// TIA Portal V17 export
// export: Created 2023-02-13T11:16:21.0492472Z, ExportSetting WithDefaults, DisplayName Totally Integrated Automation Portal, DisplayVersion V17, DisplayName TIA Portal Openness, DisplayVersion V17, DisplayName TIA Portal Teamcenter Gateway, DisplayVersion V17, DisplayName TIA Portal Version Control Interface, DisplayVersion V17, DisplayName SINAMICS Startdrive Advanced, DisplayVersion V17, DisplayName SINAMICS Startdrive G130, G150, S120, S150, SINAMICS MV, S210, DisplayVersion V17, DisplayName SINAMICS Startdrive G110M, G120, G120C, G120D, G120P, G115D, DisplayVersion V17, DisplayName STEP 7 Professional, DisplayVersion V17, DisplayName STEP 7 Safety, DisplayVersion V17, DisplayName WinCC Professional, DisplayVersion V17
DATA_BLOCK "IO_Valve_Blending_DB"   // DB8
VERSION : 0.1
// stored: AutoNumber true, DBAccessibleFromOPCUA true, DBAccessibleFromWebserver true, InstanceOfName IO_Valve_Blending, InstanceOfType FB
"IO_Valve_Blending"
   // VAR_INPUT
   //    lock : Bool;
   //    Init : Bool;
   //    Reset : Bool;
   // END_VAR
   // VAR
   //    "AV-20.01" { S7_SetPoint := 'True'} : "Valve";
   //    "AV-20.02" { S7_SetPoint := 'True'} : "Valve";
   //    "AV-20.03" { S7_SetPoint := 'True'} : "Valve";
   //    "AV-20.04" { S7_SetPoint := 'True'} : "Valve";
   //    "AV-20.05" { S7_SetPoint := 'True'} : "Valve";
   //    "AV-20.06" { S7_SetPoint := 'True'} : "Valve";
   //    "AV-20.07" { S7_SetPoint := 'True'} : "Valve";
   //    "AV-20.08" { S7_SetPoint := 'True'} : "Valve";
   //    "AV-20.09" { S7_SetPoint := 'True'} : "Valve";
   //    "AV-20.10" { S7_SetPoint := 'True'} : "Valve";
   //    "AV-20.11" { S7_SetPoint := 'True'} : "Valve";
   //    "AV-20.12" { S7_SetPoint := 'True'} : "Valve";
   //    "AV-20.13" { S7_SetPoint := 'True'} : "Valve";
   //    "AV-20.14" { S7_SetPoint := 'True'} : "Valve";
   //    "AV-20.15" { S7_SetPoint := 'True'} : "Valve";
   //    "AV-20.16" { S7_SetPoint := 'True'} : "Valve";
   //    "AV-20.17" { S7_SetPoint := 'True'} : "Valve";
   //    "AV-20.31" { S7_SetPoint := 'True'} : "Valve";
   //    "AV-20.32" { S7_SetPoint := 'True'} : "Valve";
   //    "AV-20.33" { S7_SetPoint := 'True'} : "Valve";
   //    "AV-20.34" { S7_SetPoint := 'True'} : "Valve";
   //    "AV-20.35" { S7_SetPoint := 'True'} : "Valve";
   //    "AV-20.36" { S7_SetPoint := 'True'} : "Valve";
   //    "AV-20.37" { S7_SetPoint := 'True'} : "Valve";
   //    "AV-20.38" { S7_SetPoint := 'True'} : "Valve";
   //    "AV-20.39" { S7_SetPoint := 'True'} : "Valve";
   //    "AV-20.40" { S7_SetPoint := 'True'} : "Valve";
   //    "AV-20.41" { S7_SetPoint := 'True'} : "Valve";
   //    "AV-21.01" { S7_SetPoint := 'True'} : "Valve";
   //    "AV-21.02" { S7_SetPoint := 'True'} : "Valve";
   //    "AV-21.03" { S7_SetPoint := 'True'} : "Valve";
   //    "AV-21.04" { S7_SetPoint := 'True'} : "Valve";
   //    "AV-21.05" { S7_SetPoint := 'True'} : "Valve";
   //    "AV-21.06" { S7_SetPoint := 'True'} : "Valve";
   //    "AV-21.07" { S7_SetPoint := 'True'} : "Valve";
   //    "AV-21.08" { S7_SetPoint := 'True'} : "Valve";
   //    "AV-21.09" { S7_SetPoint := 'True'} : "Valve";
   //    "AV-21.10" { S7_SetPoint := 'True'} : "Valve";
   //    "AV-21.11" { S7_SetPoint := 'True'} : "Valve";
   //    "AV-21.12" { S7_SetPoint := 'True'} : "Valve";
   //    "AV-21.13" { S7_SetPoint := 'True'} : "Valve";
   //    "AV-21.14" { S7_SetPoint := 'True'} : "Valve";
   //    "AV-21.15" { S7_SetPoint := 'True'} : "Valve";
   //    "AV-21.16" { S7_SetPoint := 'True'} : "Valve";
   //    "AV-21.17" { S7_SetPoint := 'True'} : "Valve";
   //    "AV-21.18" { S7_SetPoint := 'True'} : "Valve";
   //    "AV-21.31" { S7_SetPoint := 'True'} : "Valve";
   //    "AV-21.32" { S7_SetPoint := 'True'} : "Valve";
   //    "AV-21.33" { S7_SetPoint := 'True'} : "Valve";
   //    "AV-21.34" { S7_SetPoint := 'True'} : "Valve";
   //    "AV-21.35" { S7_SetPoint := 'True'} : "Valve";
   //    "AV-21.36" { S7_SetPoint := 'True'} : "Valve";
   //    "AV-21.37" { S7_SetPoint := 'True'} : "Valve";
   //    "AV-21.38" { S7_SetPoint := 'True'} : "Valve";
   //    "AV-21.39" { S7_SetPoint := 'True'} : "Valve";
   //    "AV-21.40" { S7_SetPoint := 'True'} : "Valve";
   //    "AV-21.41" { S7_SetPoint := 'True'} : "Valve";
   //    "AV-22.01" { S7_SetPoint := 'True'} : "Valve";
   //    "AV-22.02" { S7_SetPoint := 'True'} : "Valve";
   //    "AV-22.03" { S7_SetPoint := 'True'} : "Valve";
   //    "AV-22.06" { S7_SetPoint := 'True'} : "Valve";
   //    "AV-22.11" { S7_SetPoint := 'True'} : "Valve";
   //    "AV-22.21" { S7_SetPoint := 'True'} : "Valve";
   //    "AV-22.22" { S7_SetPoint := 'True'} : "Valve";
   //    "AV-30.01" { S7_SetPoint := 'True'} : "Valve";
   //    "AV-30.02" { S7_SetPoint := 'True'} : "Valve";
   //    "AV-30.03" { S7_SetPoint := 'True'} : "Valve";
   //    "AV-30.04" { S7_SetPoint := 'True'} : "Valve";
   //    "AV-30.05" { S7_SetPoint := 'True'} : "Valve";
   //    "AV-30.06" { S7_SetPoint := 'True'} : "Valve";
   //    "AV-30.07" { S7_SetPoint := 'True'} : "Valve";
   //    "AV-30.08" { S7_SetPoint := 'True'} : "Valve";
   //    "AV-30.09" { S7_SetPoint := 'True'} : "Valve";
   //    "AV-30.10" { S7_SetPoint := 'True'} : "Valve";
   //    "AV-30.11" { S7_SetPoint := 'True'} : "Valve";
   //    "AV-30.12" { S7_SetPoint := 'True'} : "Valve";
   //    "AV-30.13" { S7_SetPoint := 'True'} : "Valve";
   //    "AV-30.14" { S7_SetPoint := 'True'} : "Valve";
   //    "AV-30.15" { S7_SetPoint := 'True'} : "Valve";
   //    "AV-30.16" { S7_SetPoint := 'True'} : "Valve";
   //    "AV-30.17" { S7_SetPoint := 'True'} : "Valve";
   //    "AV-30.31" { S7_SetPoint := 'True'} : "Valve";
   //    "AV-30.32" { S7_SetPoint := 'True'} : "Valve";
   //    "AV-30.33" { S7_SetPoint := 'True'} : "Valve";
   //    "AV-30.34" { S7_SetPoint := 'True'} : "Valve";
   //    "AV-30.35" { S7_SetPoint := 'True'} : "Valve";
   //    "AV-30.36" { S7_SetPoint := 'True'} : "Valve";
   //    "AV-30.37" { S7_SetPoint := 'True'} : "Valve";
   //    "AV-30.38" { S7_SetPoint := 'True'} : "Valve";
   //    "AV-30.39" { S7_SetPoint := 'True'} : "Valve";
   //    "AV-30.40" { S7_SetPoint := 'True'} : "Valve";
   //    "AV-30.41" { S7_SetPoint := 'True'} : "Valve";
   //    "AV-31.01" { S7_SetPoint := 'True'} : "Valve";
   //    "AV-31.02" { S7_SetPoint := 'True'} : "Valve";
   //    "AV-31.03" { S7_SetPoint := 'True'} : "Valve";
   //    "AV-31.04" { S7_SetPoint := 'True'} : "Valve";
   //    "AV-31.05" { S7_SetPoint := 'True'} : "Valve";
   //    "AV-31.06" { S7_SetPoint := 'True'} : "Valve";
   //    "AV-31.07" { S7_SetPoint := 'True'} : "Valve";
   //    "AV-31.08" { S7_SetPoint := 'True'} : "Valve";
   //    "AV-31.09" { S7_SetPoint := 'True'} : "Valve";
   //    "AV-31.10" { S7_SetPoint := 'True'} : "Valve";
   //    "AV-31.11" { S7_SetPoint := 'True'} : "Valve";
   //    "AV-31.12" { S7_SetPoint := 'True'} : "Valve";
   //    "AV-31.13" { S7_SetPoint := 'True'} : "Valve";
   //    "AV-31.14" { S7_SetPoint := 'True'} : "Valve";
   //    "AV-31.15" { S7_SetPoint := 'True'} : "Valve";
   //    "AV-31.16" { S7_SetPoint := 'True'} : "Valve";
   //    "AV-31.17" { S7_SetPoint := 'True'} : "Valve";
   //    "AV-31.18" { S7_SetPoint := 'True'} : "Valve";
   //    "AV-31.31" { S7_SetPoint := 'True'} : "Valve";
   //    "AV-31.32" { S7_SetPoint := 'True'} : "Valve";
   //    "AV-31.33" { S7_SetPoint := 'True'} : "Valve";
   //    "AV-31.34" { S7_SetPoint := 'True'} : "Valve";
   //    "AV-31.35" { S7_SetPoint := 'True'} : "Valve";
   //    "AV-31.36" { S7_SetPoint := 'True'} : "Valve";
   //    "AV-31.37" { S7_SetPoint := 'True'} : "Valve";
   //    "AV-31.38" { S7_SetPoint := 'True'} : "Valve";
   //    "AV-31.39" { S7_SetPoint := 'True'} : "Valve";
   //    "AV-31.40" { S7_SetPoint := 'True'} : "Valve";
   //    "AV-31.41" { S7_SetPoint := 'True'} : "Valve";
   //    "AV-31.51" { S7_SetPoint := 'True'} : "Valve";
   //    "AV-31.52" { S7_SetPoint := 'True'} : "Valve";
   //    "AV-31.53" { S7_SetPoint := 'True'} : "Valve";
   //    "AV-31.54" { S7_SetPoint := 'True'} : "Valve";
   //    "AV-31.55" { S7_SetPoint := 'True'} : "Valve";
   //    "AV-31.56" { S7_SetPoint := 'True'} : "Valve";
   //    "AV-31.57" { S7_SetPoint := 'True'} : "Valve";
   //    "AV-31.58" { S7_SetPoint := 'True'} : "Valve";
   //    "AV-31.59" { S7_SetPoint := 'True'} : "Valve";
   //    "AV-31.60" { S7_SetPoint := 'True'} : "Valve";
   //    "AV-31.61" { S7_SetPoint := 'True'} : "Valve";
   //    "AV-31.62" { S7_SetPoint := 'True'} : "Valve";
   //    "AV-32.01" { S7_SetPoint := 'True'} : "Valve";
   //    "AV-32.02" { S7_SetPoint := 'True'} : "Valve";
   //    "AV-32.03" { S7_SetPoint := 'True'} : "Valve";
   //    "AV-32.06" { S7_SetPoint := 'True'} : "Valve";
   //    "AV-32.11" { S7_SetPoint := 'True'} : "Valve";
   //    "AV-32.21" { S7_SetPoint := 'True'} : "Valve";
   //    "AV-32.22" { S7_SetPoint := 'True'} : "Valve";
   //    "AV-20.42" { S7_SetPoint := 'True'} : "Valve";
   //    "AV-21.42" { S7_SetPoint := 'True'} : "Valve";
   //    "AV-22.04" { S7_SetPoint := 'True'} : "Valve";
   //    "AV-22.05" { S7_SetPoint := 'True'} : "Valve";
   //    "AV-30.42" { S7_SetPoint := 'True'} : "Valve";
   //    "AV-31.42" { S7_SetPoint := 'True'} : "Valve";
   //    "AV-32.04" { S7_SetPoint := 'True'} : "Valve";
   //    "AV-32.05" { S7_SetPoint := 'True'} : "Valve";
   // END_VAR
BEGIN
   "AV-20.02".OPdwCmd := 16#0008_0000;
   "AV-20.03".OPdwCmd := 16#0008_0000;
   "AV-20.04".OPdwCmd := 16#0008_0000;
   "AV-20.05".OPdwCmd := 16#0008_0000;
   "AV-20.06".OPdwCmd := 16#0008_0000;
   "AV-20.07".OPdwCmd := 16#0008_0000;
   "AV-20.08".OPdwCmd := 16#0008_0000;
   "AV-20.09".OPdwCmd := 16#0008_0000;
   "AV-20.10".OPdwCmd := 16#0008_0000;
   "AV-20.11".OPdwCmd := 16#0008_0000;
   "AV-20.12".OPdwCmd := 16#0008_0000;
   "AV-20.13".OPdwCmd := 16#0008_0000;
   "AV-20.14".OPdwCmd := 16#0008_0000;
   "AV-20.15".OPdwCmd := 16#0008_0000;
   "AV-20.16".OPdwCmd := 16#0008_0000;
   "AV-20.17".OPdwCmd := 16#0008_0000;
   "AV-20.31".OPdwCmd := 16#0008_0000;
   "AV-20.32".OPdwCmd := 16#0008_0000;
   "AV-20.33".OPdwCmd := 16#0008_0000;
   "AV-20.34".OPdwCmd := 16#0008_0000;
   "AV-20.35".OPdwCmd := 16#0008_0000;
   "AV-20.36".OPdwCmd := 16#0008_0000;
   "AV-20.37".OPdwCmd := 16#0008_0000;
   "AV-20.38".OPdwCmd := 16#0008_0000;
   "AV-20.39".OPdwCmd := 16#0008_0000;
   "AV-20.40".OPdwCmd := 16#0008_0000;
   "AV-20.41".OPdwCmd := 16#0008_0000;
   "AV-21.01".OPdwCmd := 16#0008_0000;
   "AV-21.02".OPdwCmd := 16#0008_0000;
   "AV-21.03".OPdwCmd := 16#0008_0000;
   "AV-21.04".OPdwCmd := 16#0008_0000;
   "AV-21.05".OPdwCmd := 16#0008_0000;
   "AV-21.06".OPdwCmd := 16#0008_0000;
   "AV-21.07".OPdwCmd := 16#0008_0000;
   "AV-21.08".OPdwCmd := 16#0008_0000;
   "AV-21.09".OPdwCmd := 16#0008_0000;
   "AV-21.10".OPdwCmd := 16#0008_0000;
   "AV-21.11".OPdwCmd := 16#0008_0000;
   "AV-21.12".OPdwCmd := 16#0008_0000;
   "AV-21.13".OPdwCmd := 16#0008_0000;
   "AV-21.14".OPdwCmd := 16#0008_0000;
   "AV-21.15".OPdwCmd := 16#0008_0000;
   "AV-21.16".OPdwCmd := 16#0008_0000;
   "AV-21.17".OPdwCmd := 16#0008_0000;
   "AV-21.18".OPdwCmd := 16#0008_0000;
   "AV-21.31".OPdwCmd := 16#0008_0000;
   "AV-21.32".OPdwCmd := 16#0008_0000;
   "AV-21.33".OPdwCmd := 16#0008_0000;
   "AV-21.34".OPdwCmd := 16#0008_0000;
   "AV-21.35".OPdwCmd := 16#0008_0000;
   "AV-21.36".OPdwCmd := 16#0008_0000;
   "AV-21.37".OPdwCmd := 16#0008_0000;
   "AV-21.38".OPdwCmd := 16#0008_0000;
   "AV-21.39".OPdwCmd := 16#0008_0000;
   "AV-21.40".OPdwCmd := 16#0008_0000;
   "AV-21.41".OPdwCmd := 16#0008_0000;
   "AV-22.01".OPdwCmd := 16#0008_0000;
   "AV-22.02".OPdwCmd := 16#0008_0000;
   "AV-22.03".OPdwCmd := 16#0008_0000;
   "AV-22.06".OPdwCmd := 16#0008_0000;
   "AV-22.11".OPdwCmd := 16#0008_0000;
   "AV-22.21".OPdwCmd := 16#0008_0000;
   "AV-22.22".OPdwCmd := 16#0008_0000;
   "AV-30.01".OPdwCmd := 16#0008_0000;
   "AV-30.02".OPdwCmd := 16#0008_0000;
   "AV-30.03".OPdwCmd := 16#0008_0000;
   "AV-30.04".OPdwCmd := 16#0008_0000;
   "AV-30.05".OPdwCmd := 16#0008_0000;
   "AV-30.06".OPdwCmd := 16#0008_0000;
   "AV-30.07".OPdwCmd := 16#0008_0000;
   "AV-30.08".OPdwCmd := 16#0008_0000;
   "AV-30.09".OPdwCmd := 16#0008_0000;
   "AV-30.10".OPdwCmd := 16#0008_0000;
   "AV-30.11".OPdwCmd := 16#0008_0000;
   "AV-30.12".OPdwCmd := 16#0008_0000;
   "AV-30.13".OPdwCmd := 16#0008_0000;
   "AV-30.14".OPdwCmd := 16#0008_0000;
   "AV-30.15".OPdwCmd := 16#0008_0000;
   "AV-30.16".OPdwCmd := 16#0008_0000;
   "AV-30.17".OPdwCmd := 16#0008_0000;
   "AV-30.31".OPdwCmd := 16#0008_0000;
   "AV-30.32".OPdwCmd := 16#0008_0000;
   "AV-30.33".OPdwCmd := 16#0008_0000;
   "AV-30.34".OPdwCmd := 16#0008_0000;
   "AV-30.35".OPdwCmd := 16#0008_0000;
   "AV-30.36".OPdwCmd := 16#0008_0000;
   "AV-30.37".OPdwCmd := 16#0008_0000;
   "AV-30.38".OPdwCmd := 16#0008_0000;
   "AV-30.39".OPdwCmd := 16#0008_0000;
   "AV-30.40".OPdwCmd := 16#0008_0000;
   "AV-30.41".OPdwCmd := 16#0008_0000;
   "AV-31.01".OPdwCmd := 16#0008_0000;
   "AV-31.02".OPdwCmd := 16#0008_0000;
   "AV-31.03".OPdwCmd := 16#0008_0000;
   "AV-31.04".OPdwCmd := 16#0008_0000;
   "AV-31.05".OPdwCmd := 16#0008_0000;
   "AV-31.06".OPdwCmd := 16#0008_0000;
   "AV-31.07".OPdwCmd := 16#0008_0000;
   "AV-31.08".OPdwCmd := 16#0008_0000;
   "AV-31.09".OPdwCmd := 16#0008_0000;
   "AV-31.10".OPdwCmd := 16#0008_0000;
   "AV-31.11".OPdwCmd := 16#0008_0000;
   "AV-31.12".OPdwCmd := 16#0008_0000;
   "AV-31.13".OPdwCmd := 16#0008_0000;
   "AV-31.14".OPdwCmd := 16#0008_0000;
   "AV-31.15".OPdwCmd := 16#0008_0000;
   "AV-31.16".OPdwCmd := 16#0008_0000;
   "AV-31.17".OPdwCmd := 16#0008_0000;
   "AV-31.18".OPdwCmd := 16#0008_0000;
   "AV-31.31".OPdwCmd := 16#0008_0000;
   "AV-31.32".OPdwCmd := 16#0008_0000;
   "AV-31.33".OPdwCmd := 16#0008_0000;
   "AV-31.34".OPdwCmd := 16#0008_0000;
   "AV-31.35".OPdwCmd := 16#0008_0000;
   "AV-31.36".OPdwCmd := 16#0008_0000;
   "AV-31.37".OPdwCmd := 16#0008_0000;
   "AV-31.38".OPdwCmd := 16#0008_0000;
   "AV-31.39".OPdwCmd := 16#0008_0000;
   "AV-31.40".OPdwCmd := 16#0008_0000;
   "AV-31.41".OPdwCmd := 16#0008_0000;
   "AV-31.51".OPdwCmd := 16#0008_0000;
   "AV-31.52".OPdwCmd := 16#0008_0000;
   "AV-31.53".OPdwCmd := 16#0008_0000;
   "AV-31.54".OPdwCmd := 16#0008_0000;
   "AV-31.55".OPdwCmd := 16#0008_0000;
   "AV-31.56".OPdwCmd := 16#0008_0000;
   "AV-31.57".OPdwCmd := 16#0008_0000;
   "AV-31.58".OPdwCmd := 16#0008_0000;
   "AV-31.59".OPdwCmd := 16#0008_0000;
   "AV-31.60".OPdwCmd := 16#0008_0000;
   "AV-31.61".OPdwCmd := 16#0008_0000;
   "AV-31.62".OPdwCmd := 16#0008_0000;
   "AV-32.01".OPdwCmd := 16#0008_0000;
   "AV-32.02".OPdwCmd := 16#0008_0000;
   "AV-32.03".OPdwCmd := 16#0008_0000;
   "AV-32.06".OPdwCmd := 16#0008_0000;
   "AV-32.11".OPdwCmd := 16#0008_0000;
   "AV-32.21".OPdwCmd := 16#0008_0000;
   "AV-32.22".OPdwCmd := 16#0008_0000;
   "AV-20.42".OPdwCmd := 16#0008_0000;
   "AV-21.42".OPdwCmd := 16#0008_0000;
   "AV-22.04".OPdwCmd := 16#0008_0000;
   "AV-22.05".OPdwCmd := 16#0008_0000;
   "AV-30.42".OPdwCmd := 16#0008_0000;
   "AV-31.42".OPdwCmd := 16#0008_0000;
   "AV-32.04".OPdwCmd := 16#0008_0000;
   "AV-32.05".OPdwCmd := 16#0008_0000;
END_DATA_BLOCK
